TYPE ST_Path :
STRUCT
	startPath : INT;
	endPath : INT;
END_STRUCT
END_TYPE

(* stored: Version 1.1.0.1
   DUT ST_Path: Id {9f922bcd-f4c5-4d35-8e0d-8eda12194373} *)
